Staubli VAL3: getList.pgx

program getList(string x_sPtPara, string& x_sOutPtpara[])
  local num l_nRes
  local num l_ni
begin
  //对参数x_sPtPara进行解析，得到相应信息

  call PublicProg:SplitChar(l_nRes,x_sPtPara,"/",x_sOutPtpara)

end
